// TIA Portal V20 export
DATA_BLOCK "DB_Alarm"   // DB14
// stored: Access Published, MemoryReserve 100, Namespace EmptyLine
   VAR
      "word" : Struct
         Line : Struct
            EmptyLine : Struct
               Conveyor : Array[_.minEmptyLine.._.maxEmptyLine] of Word;
            END_STRUCT;
         END_STRUCT;
      END_STRUCT;
      Simu : Word;
   END_VAR
BEGIN
END_DATA_BLOCK
